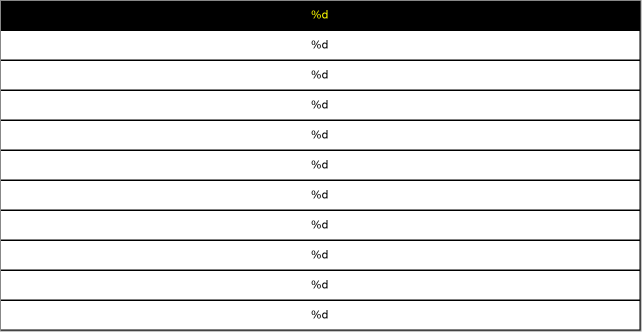
VISUALIZATION TWISTED_CUPS_SHIFT_ELEMENT  // 642x332
VAR_INPUT
	index:		UDINT;
END_VAR
    Rectangle (0,0 640x30), "%d", text variable: wu_twistedCups_shiftRegister_debug.outer_shift_debug[90+index].step_id
    Rectangle (0,30 640x30), "%d", text variable: wu_twistedCups_shiftRegister_debug.outer_shift_debug[90+index].status.0, colour toggle: wu_twistedCups_shiftRegister_debug.outer_shift_debug[90+index].status.0
    Rectangle (0,90 640x30), "%d", text variable: wu_twistedCups_shiftRegister_debug.outer_shift_debug[90+index].reject_reason
    Rectangle (0,150 640x30), "%d", text variable: wu_twistedCups_shiftRegister_debug.outer_shift_debug[90+index].status.3, colour toggle: wu_twistedCups_shiftRegister_debug.outer_shift_debug[90+index].status.3
    Rectangle (0,210 640x30), "%d", text variable: wu_twistedCups_shiftRegister_debug.outer_shift_debug[90+index].product_id
    Rectangle (0,60 640x30), "%d", text variable: wu_twistedCups_shiftRegister_debug.inner_shift_debug[90+index].status.0, colour toggle: wu_twistedCups_shiftRegister_debug.inner_shift_debug[90+index].status.0
    Rectangle (0,120 640x30), "%d", text variable: wu_twistedCups_shiftRegister_debug.inner_shift_debug[90+index].reject_reason
    Rectangle (0,180 640x30), "%d", text variable: wu_twistedCups_shiftRegister_debug.inner_shift_debug[90+index].status.3, colour toggle: wu_twistedCups_shiftRegister_debug.inner_shift_debug[90+index].status.3
    Rectangle (0,240 640x30), "%d", text variable: wu_twistedCups_shiftRegister_debug.inner_shift_debug[90+index].product_id
    Rectangle (0,270 640x30), "%d", text variable: wu_twistedCups_shiftRegister_debug.outer_shift_debug[90+index].robot_id
    Rectangle (0,300 640x30), "%d", text variable: wu_twistedCups_shiftRegister_debug.inner_shift_debug[90+index].robot_id
END_VISUALIZATION

(* stored: Version 1.1.0.1, ProductVersion 3.1.4024.3
   Visu TWISTED_CUPS_SHIFT_ELEMENT: Id {fc513f34-434b-43f3-893b-1605676c9834} *)
